TYPE ID : STRING(10); END_TYPE

(* stored: Version 1.1.0.1
   DUT ID: Id {257580b0-f66a-0734-1d29-19d853047497} *)
